KUKA KRL data list: Int_Tooling.dat

&ACCESS RVO2
&REL 18
&PARAM DISKPATH = KRC:\R1\HG_Mes
DEFDAT  INT_TOOLING PUBLIC

GLOBAL BOOL Grip_1=FALSE ; ????1???? ????????1
GLOBAL BOOL Grip_2=FALSE ; ????2???? ????????2
BOOL Grip_OK=FALSE ;
BOOL Grip_Reset=FALSE

BOOL Button_1_On=FALSE
BOOL Button_1_Up=FALSE
BOOL Button_2_On=FALSE
BOOL Button_2_Up=FALSE
GLOBAL BOOL Reset_Tooling=FALSE ; ????????????????

ENDDAT
